    PROC MoveGridDatum()
        !Sweep across bed maintaining Z height through offsets
        FOR j FROM 9 TO 4 DO
            FOR k FROM 11 TO 1 DO
                !Move x
                PlotBedGrid(k*XGridSpacing+100),(j*YGridSpacing+100),Bed1Zread{10-j,(k+1)};
            ENDFOR
        ENDFOR
    ENDPROC


    PROC VacuumBed()

        VAR num VacOverlap:=-400;
        IF ToolNum<>5 THEN
            Home;
            Vac_Pickup;
        ELSE
            CurrentJoints:=CJointT();
            CurrentPos:=CalcRobT(CurrentJoints,tVac\WObj:=Bed1Wyong);
            IF CurrentPos.trans.x<0 AND (CurrentPos.trans.z<150) THEN
                MoveL Offs(CurrentPos,0,0,(150-CurrentPos.trans.z)),v500,z5,tVac\WObj:=Bed1Wyong;
            ELSEIF (CurrentPos.trans.z<700) THEN
                MoveL Offs(CurrentPos,0,0,(700-CurrentPos.trans.z)),v500,z5,tVac\WObj:=Bed1Wyong;
            ENDIF
        ENDIF

        pTemp:=pVacStart;
        pTemp2:=pVacStart;
        pTemp2.trans.x:=pVacStart2.trans.x;
        pTemp2.extax.eax_a:=pVacStart2.extax.eax_a;

        Vac_on;
        FOR i FROM 0 TO (Round((pVacStart.trans.y-pVacStart2.trans.y)/(-1*VacOverlap))) DO
            IF pTemp.trans.y+i*VacOverlap>pVacStart2.trans.y THEN
                MoveJ Offs(pTemp,0,i*VacOverlap,150),v500,z5,tVac\WObj:=Bed1Wyong;
                MoveL Offs(pTemp,0,i*VacOverlap,0),v50,z5,tVac\WObj:=Bed1Wyong;
                MoveL Offs(pTemp2,0,i*VacOverlap,0),v100,z5,tVac\WObj:=Bed1Wyong;
                MoveL Offs(pTemp2,0,i*VacOverlap,150),v50,fine,tVac\WObj:=Bed1Wyong;
            ENDIF
        ENDFOR

        Vac_off;

        CurrentJoints:=CJointT();
        CurrentPos:=CalcRobT(CurrentJoints,tVac\WObj:=wobj0);
        MoveL Offs(CurrentPos,0,0,800-CurrentPos.trans.z),v100,z5,tVac\WObj:=wobj0;

    ENDPROC

    PROC JointPositions()

        VAR num PolishOverlap:=450;
        pPolTemp:=pPolStart1;
        pPolTemp2:=pPolStart1;
        pPolTemp2.extax.eax_a:=pPolStart1.extax.eax_a-7500;
        pPolTemp2.trans.x:=-7500;

        pPolTemp.rot:=pPolStart1.rot;
        pPolTemp2.rot:=pPolStart1.rot;

        pPolTemp2.rot:=pPolStart2.rot;
        pPolTemp2.extax.eax_a:=pPolStart1.extax.eax_a-8500;
        CurrentJoints5:=CJointT();
        CurrentJoints6:=CalcJointT(Offs(pPolTemp2,50,(1+1)*PolishOverlap,40),tPolish\WObj:=Bed1Wyong);

    ENDPROC


    PROC RobbiePlot()

        ! !Write R
        !PlotLine 6900,1000, 6900,2000;
        !PlotArc 6900,2000,6650,1750,6900,1500;
        !PlotLine 6900,1500,6650,1000;

        !!Write O
        !PlotArc 6300,2000, 6050,1500,6300,1000;
        !PlotArc 6300,1000, 6550,1500,6300,2000;

        !!Write B
        !PlotLine 5700,1000, 5700,2000;
        !PlotArc 5700,2000,5450,1750,5700,1500;
        !PlotArc 5700,1500,5450,1250,5700,1000;

        !!Write B
        !PlotLine 5100,1000, 5100,2000;
        !PlotArc 5100,2000,4850,1750,5100,1500;
        !PlotArc 5100,1500,4850,1250,5100,1000;

        !!Write I
        !PlotLine 4500,1000, 4500,2000;

        !!Write E
        !PlotLine 3900,1000, 3900,2000;
        !PlotLine 3900,2000, 3400,2000;
        !PlotLine 3900,1500, 3400,1500;
        !PlotLine 3900,1000, 3400,1000;

        !formbox
        PlotRect 2000,500,2000,3500,6000,3500,6000,500;
        !Ferrule
        WaitTime\inpos,0.1;
        PlotCirc 2250,750,(PlotCircleD/2);
        PlotLine(2250-PlotCircleD/2-CrossHairExt),750,(2250+PlotCircleD/2+CrossHairExt),750;
        PlotLine 2250,(750-PlotCircleD/2-CrossHairExt),2250,(750+PlotCircleD/2+CrossHairExt);
        !Ferrule
        WaitTime\inpos,0.1;
        PlotCirc 2250,3250,(PlotCircleD/2);
        PlotLine(2250-PlotCircleD/2-CrossHairExt),3250,(2250+PlotCircleD/2+CrossHairExt),3250;
        PlotLine 2250,(3250-PlotCircleD/2-CrossHairExt),2250,(3250+PlotCircleD/2+CrossHairExt);
        !Grout tube Casee 4
        WaitTime\inpos,0.1;
        iCoord1x:=6000;
        iCoord1y:=2000;
        iAngle:=0;
        PlotRect iCoord1x-GroutWidth/2*Sin(iAngle)-GroutHeight*Cos(iAngle),iCoord1y+GroutHeight*Sin(iAngle)-GroutWidth/2*Cos(iAngle),iCoord1x+GroutWidth/2*Sin(iAngle)-GroutHeight*Cos(iAngle),iCoord1y+GroutHeight*Sin(iAngle)+GroutWidth/2*Cos(iAngle),iCoord1x+GroutWidth/2*Sin(iAngle),iCoord1y+GroutWidth/2*Cos(iAngle),iCoord1x-GroutWidth/2*Sin(iAngle),iCoord1y-GroutWidth/2*Cos(iAngle);

        !Lifting points 180 angle
        WaitTime\inpos,0.1;
        TriangleAngle:=180;
        iCoord1x:=5000;
        iCoord1y:=3500;
        PlotLine iCoord1x-TriangleHeight*Sin(TriangleAngle),iCoord1y-TriangleHeight*Cos(TriangleAngle),iCoord1x-TriangleBase/2*Cos(TriangleAngle),iCoord1y+TriangleBase/2*Sin(TriangleAngle);
        PlotLine iCoord1x-TriangleBase/2*Cos(TriangleAngle),iCoord1y+TriangleBase/2*Sin(TriangleAngle),iCoord1x+TriangleBase/2*Cos(TriangleAngle),iCoord1y-TriangleBase/2*Sin(TriangleAngle);
        PlotLine iCoord1x+TriangleBase/2*Cos(TriangleAngle),iCoord1y-TriangleBase/2*Sin(TriangleAngle),iCoord1x-TriangleHeight*Sin(TriangleAngle),iCoord1y-TriangleHeight*Cos(TriangleAngle);
        !Lifting points 180 angle
        WaitTime\inpos,0.1;
        TriangleAngle:=180;
        iCoord1x:=3000;
        iCoord1y:=3500;
        PlotLine iCoord1x-TriangleHeight*Sin(TriangleAngle),iCoord1y-TriangleHeight*Cos(TriangleAngle),iCoord1x-TriangleBase/2*Cos(TriangleAngle),iCoord1y+TriangleBase/2*Sin(TriangleAngle);
        PlotLine iCoord1x-TriangleBase/2*Cos(TriangleAngle),iCoord1y+TriangleBase/2*Sin(TriangleAngle),iCoord1x+TriangleBase/2*Cos(TriangleAngle),iCoord1y-TriangleBase/2*Sin(TriangleAngle);
        PlotLine iCoord1x+TriangleBase/2*Cos(TriangleAngle),iCoord1y-TriangleBase/2*Sin(TriangleAngle),iCoord1x-TriangleHeight*Sin(TriangleAngle),iCoord1y-TriangleHeight*Cos(TriangleAngle);

        Plotter_Dropoff;

    ENDPROC

    PROC PolishDemo()
        IF ToolNum<>6 THEN
            Home;
            Polish_Pickup;
        ELSE
            CurrentJoints:=CJointT();
            CurrentPos:=CalcRobT(CurrentJoints,tPolish\WObj:=wobj0);
            IF CurrentPos.trans.z<600 THEN
                MoveL Offs(CurrentPos,0,0,(600-CurrentPos.trans.z)),v500,z5,tPolish;
            ENDIF
        ENDIF
        MoveJ pPolHome,v500,z5,tPolish;
        pPolTemp:=pPolStart1;
        pPolTemp2:=pPolStart1;
        pPolTemp2.extax.eax_a:=pPolStart1.extax.eax_a-7500;
        pPolTemp2.trans.x:=-7500;
        pPolTemp.rot:=pPolStart1.rot;
        pPolTemp2.rot:=pPolStart1.rot;
        FCCalib PolishLoad;
        pPolTemp.extax.eax_a:=pPolStart1.extax.eax_a;
        MoveJ Offs(pPolTemp,0,0,100),v500,z5,tPolish\WObj:=Bed1Wyong;
        Pol_on;
        MoveL Offs(pPolTemp,0,0,50),v100,fine,tPolish\WObj:=Bed1Wyong;
        myForceVector:=FCGetForce(\Tool:=tPolish);
        FCPress1LStart Offs(pPolTemp,-25,0,55),v10,\Fz:=120,15,\ForceChange:=50\PosSupvDist:=125,z5,tPolish\WObj:=Bed1Wyong;
        pPolTemp2.extax.eax_a:=pPolStart2.extax.eax_a-300;
        FCPressL Offs(pPolTemp2,-300,0,-15),v100,130,fine,tPolish\WObj:=Bed1Wyong;
        FCPressEnd Offs(pPolTemp2,-300,0,75),v50,\DeactOnly,tPolish\WObj:=Bed1Wyong;
        CurrentJoints:=CJointT();
        CurrentPos:=CalcRobT(CurrentJoints,tPolish\WObj:=Bed1Wyong);
        MoveJ Offs(Reltool(CurrentPos,0,0,-100),0,450,0),v100,fine,tPolish\WObj:=Bed1Wyong;
        Pol_off;
        Polish_Dropoff;
    ENDPROC



    PROC BedGrid()

        !        MoveJ Offs(p10Maps,500*(1-1)+2000*(1-1),650*(1-1),50),v500,z5,tTCMaster\WObj:=Bed1Wyong;
        !        MoveL Offs(p10Maps,500*(1-1)+2000*(1-1),650*(1-1),0),v500,fine,tTCMaster\WObj:=Bed1Wyong;
        !        Stop;
        !        MoveL Offs(p10Maps,500*(1-1)+2000*(1-1),650*(1-1),50),v500,z5,tTCMaster\WObj:=Bed1Wyong;
        !        Stop;

        FOR i FROM 1 TO 5 DO
            !Move EAX
            FOR k FROM 1 TO 4 DO
                !Move x
                FOR j FROM 1 TO 4 DO
                    !Move y
                    IF 500*(k-1)+2000*(i-1)<8001 THEN
                        p10maps.extax.eax_a:=Bed1Wyong.uframe.trans.x+p10Maps.trans.x-500*(k-1)-2000*(i-1);
                        IF p10maps.extax.eax_a>10150 THEN
                            p10maps.extax.eax_a:=10100;
                        ENDIF
                        IF p10maps.extax.eax_a<1000 THEN
                            p10maps.extax.eax_a:=1000;
                        ENDIF

                        !MoveJ Offs(p10Maps,-500*(k-1)-2000*(i-1),650*(j-1),50),v500,z5,tTCMaster\WObj:=Bed1Wyong;
                        !MoveL Offs(p10Maps,-500*(k-1)-2000*(i-1),650*(j-1),0),v500,fine,tTCMaster\WObj:=Bed1Wyong;
                        !TPReadNum BedZread,"Enter Z reading";
                        !BedZreads{5-j,((i-1)*4+k)}:=BedZread;
                        BedZpos{5-j,((i-1)*4+k),1}:=p10Maps.trans.x-500*(k-1)-2000*(i-1);
                        BedZpos{5-j,((i-1)*4+k),2}:=p10maps.trans.y+650*(j-1);
                        !MoveL Offs(p10Maps,-500*(k-1)-2000*(i-1),650*(j-1),50),v500,z5,tTCMaster\WObj:=Bed1Wyong;
                    ENDIF

                ENDFOR
            ENDFOR
        ENDFOR
        Stop;

    ENDPROC


    PROC ClearBedZ()

        FOR i FROM 1 TO 4 DO
            !Move EAX
            FOR k FROM 1 TO 24 DO
                !Move x
                BedZreads{i,k}:=0;
                BedZpos{i,k,1}:=0;
                BedZpos{i,k,2}:=0;
            ENDFOR
        ENDFOR

    ENDPROC




    PROC BHTestTask()
        TPErase;
        TPWrite "BH Test Task";
        TPWrite "Press Play to confirm and start task";
        Stop;

        TPErase;
        TPWrite "Starting BH Test Task...";

        Heli_Pickup;
        MoveJ Offs(ptHeli,0,0,1000),v500,fine,tHeli;
        TPWrite "Helicopter tool at 1000mm above pickup";
        WaitTime 2;

        Heli_Dropoff;
        TPWrite "Helicopter tool dropped off";

        Polish_Pickup;
        MoveJ Offs(ptPolish,0,0,1000),v500,fine,tPolish;
        TPWrite "Polisher tool at 1000mm above pickup";
        WaitTime 2;

        Polish_Dropoff;
        TPWrite "Polisher tool dropped off";

        Home;
        TPWrite "BH Test Task Complete";

    ERROR
        RAISE ;
    ENDPROC



    PROC Datum()
        ! Datum - draws small circle at Bed1Wyong origin (0,0)
        ! Generated by Onyx Toolpath Generator
        VAR robtarget pDatumCenter;
        VAR robtarget pDatumCircle;
        VAR num DatumZ:=300;
        VAR num DatumRadius:=100;
        VAR num SafeZ:=500;
        VAR num i;

        TPWrite "Datum: ToolNum=" \Num:=ToolNum;
        IF ToolNum<>4 THEN
            TPWrite "No plotter! Will pickup plotter.";
            Stop;
            Home;
            Plotter_Pickup;
        ELSE
            CurrentJoints:=CJointT();
            CurrentPos:=CalcRobT(CurrentJoints,tPlotter\WObj:=wobj0);
            IF CurrentPos.trans.z<600 THEN
                MoveL Offs(CurrentPos,0,0,(600-CurrentPos.trans.z)),v500,z5,tPlotter;
            ENDIF
        ENDIF

        ConfL\Off;
        ConfJ\Off;

        pDatumCenter:=[[0,0,DatumZ],[0,0,1,0],[0,0,0,0],[0,9E+09,9E+09,9E+09,9E+09,9E+09]];
        pDatumCenter.rot:=OrientZYX(-90,0,180);
        pDatumCenter.extax.eax_a:=6500;

        TPWrite "Datum: Drawing circle at origin";
        TPWrite "Press Play to continue";
        Stop;

        pDatumCircle:=pDatumCenter;
        pDatumCircle.trans.z:=SafeZ;
        MoveJ pDatumCircle,v500,z5,tPlotter\WObj:=Bed1Wyong;

        pDatumCircle.trans.x:=DatumRadius;
        pDatumCircle.trans.z:=DatumZ;
        MoveJ pDatumCircle,v500,z5,tPlotter\WObj:=Bed1Wyong;

        FOR i FROM 1 TO 8 DO
            pDatumCircle.trans.x:=DatumRadius*Cos(i*45);
            pDatumCircle.trans.y:=DatumRadius*Sin(i*45);
            MoveJ pDatumCircle,v100,fine,tPlotter\WObj:=Bed1Wyong;
        ENDFOR

        pDatumCircle.trans.x:=0;
        pDatumCircle.trans.y:=0;
        pDatumCircle.trans.z:=DatumZ;
        MoveJ pDatumCircle,v100,fine,tPlotter\WObj:=Bed1Wyong;

        TPWrite "Plotter at datum center (0,0)";
        TPWrite "Press Play to return tool";
        Stop;

        pDatumCircle.trans.z:=SafeZ;
        MoveJ pDatumCircle,v500,z5,tPlotter\WObj:=Bed1Wyong;

        ConfL\On;
        ConfJ\On;

        Plotter_Dropoff;
        Home;

        TPWrite "Datum Complete";
    ERROR
        RAISE;
    ENDPROC


    PROC PyHeli()
        ! PyHeli - Helicopter serpentine pattern
        ! Workzone: panel
        ! Force Control DISABLED (dummy run)
        ! Generated by Onyx Toolpath Generator

        VAR robtarget pHeliPos;
        VAR robtarget pHeliEnd;
        VAR num HeliZ:=450;
        VAR num SafeZ:=500;

        ! Workspace bounds (with offsets applied)
        VAR num WorkMinX:=2200;
        VAR num WorkMaxX:=7850;
        VAR num WorkMinY:=200;
        VAR num WorkMaxY:=2200;

        ! Pattern parameters
        VAR num StepSize:=450;
        VAR num SweepDir:=1;
        VAR num StepDir:=-1;
        VAR num CurrentY:=2200;
        VAR num CurrentX:=2200;
        VAR num NextY;
        VAR num NextX;
        VAR num StartX;
        VAR num EndX;
        VAR num StartY;
        VAR num EndY;

        ! Speed and blade parameters
        VAR num HeliSpeed:=100;
        VAR num HeliAngle:=1;
        VAR speeddata vHeliTravel:=[500,15,2000,15];
        VAR num NumPasses;
        ! Force control disabled

        NumPasses:=Trunc(Abs(WorkMaxY-WorkMinY)/StepSize)+1;

        TPWrite "PyHeli: Serpentine Pattern";
        TPWrite "Work Area (7850,2200) to (2200,200)";
        TPWrite "Passes=" \Num:=NumPasses;
        TPWrite "Step=" \Num:=StepSize;
        TPWrite "Force=OFF (dummy)";

        IF ToolNum<>2 THEN
            TPWrite "PyHeli: ToolNum<>2, need pickup";
            Stop;
            Home;
            Heli_Pickup;
        ELSE
            CurrentJoints:=CJointT();
            CurrentPos:=CalcRobT(CurrentJoints,tHeli\WObj:=Bed1Wyong);
            IF CurrentPos.trans.z<SafeZ THEN
                MoveL Offs(CurrentPos,0,0,(SafeZ-CurrentPos.trans.z)),v500,z5,tHeli\WObj:=Bed1Wyong;
            ENDIF
        ENDIF

        ! Set start/end based on sweep direction
        IF SweepDir=1 THEN
            StartX:=WorkMinX;
            EndX:=WorkMaxX;
        ELSE
            StartX:=WorkMaxX;
            EndX:=WorkMinX;
        ENDIF

        ! Set initial position with fixed orientation
        pHeliPos:=[[0,0,HeliZ],OrientZYX(0,0,180),[0,0,0,0],[0,9E+09,9E+09,9E+09,9E+09,9E+09]];

        ! Move to row start above surface (HOVER)
        pHeliPos.trans.x:=-StartX;
        pHeliPos.trans.y:=CurrentY;
        pHeliPos.trans.z:=SafeZ;
        pHeliPos.extax.eax_a:=Bed1Wyong.uframe.trans.x-StartX;
        MoveJ pHeliPos,v500,z5,tHeli\WObj:=Bed1Wyong;

        ! Disable configuration tracking for serpentine movements
        ConfL\Off;
        ConfJ\Off;

        ! Home stepper before setting blade angle (ensures StepperPos is valid)
        TPWrite "Homing blade stepper...";
        Heli_Stepper_Home;
        TPWrite "Stepper homed";

        ! Set blade angle while hovering
        TPWrite "Setting blade angle to " \Num:=HeliAngle;
        HeliBlade_Angle HeliAngle;
        WaitTime 2;
        TPWrite "Blade angle set";

        ! No force calibration needed

        TPWrite "Hovering over workspace - Press Play to start";
        Stop;

        ! Start blade rotation BEFORE lowering
        TPWrite "Starting blade rotation...";
        HeliBladeSpeed HeliSpeed,"FWD";
        WaitTime 1;

        ! Lower to working height
        TPWrite "Lowering to work surface...";
        pHeliPos.trans.z:=HeliZ;
        MoveL pHeliPos,v50,fine,tHeli\WObj:=Bed1Wyong;

        ! No force control - dummy run

        ! Set up end position for first sweep
        pHeliEnd:=pHeliPos;
        pHeliEnd.trans.x:=-EndX;
        pHeliEnd.extax.eax_a:=Bed1Wyong.uframe.trans.x-EndX;

        ! ========== PASS 1: X-direction sweeps (stepping in Y) ===========
        WHILE TRUE DO
            ! === SWEEP X (full length) ===
            MoveL pHeliEnd,vHeliTravel,fine,tHeli\WObj:=Bed1Wyong;

            ! No force ramping in dummy mode

            ! Calculate next row
            NextY:=CurrentY+(StepDir*StepSize);

            ! Check if pass complete
            IF (StepDir=1 AND NextY>WorkMaxY) OR (StepDir=-1 AND NextY<WorkMinY) THEN
                EXIT;
            ENDIF

            ! Clamp to bounds
            IF NextY>WorkMaxY THEN
                NextY:=WorkMaxY;
            ELSEIF NextY<WorkMinY THEN
                NextY:=WorkMinY;
            ENDIF

            ! Step to next Y row
            pHeliEnd.trans.y:=NextY;
            MoveL pHeliEnd,vHeliTravel,fine,tHeli\WObj:=Bed1Wyong;
            CurrentY:=NextY;

            ! Flip sweep direction
            SweepDir:=-SweepDir;
            IF SweepDir=1 THEN
                StartX:=WorkMinX;
                EndX:=WorkMaxX;
            ELSE
                StartX:=WorkMaxX;
                EndX:=WorkMinX;
            ENDIF

            ! Set up end position for next sweep
            pHeliEnd.trans.x:=-EndX;
            pHeliEnd.extax.eax_a:=Bed1Wyong.uframe.trans.x-EndX;
        ENDWHILE

        ! ========== PASS 2: Y-direction sweeps (stepping in X) ==========
        TPWrite "=== PASS 2 START ===";

        ! Reset for Y-direction passes - start from current position
        CurrentX:=Abs(pHeliEnd.trans.x);
        TPWrite "Pass2: CurrentX=" \Num:=CurrentX;
        TPWrite "Pass2: CurrentY=" \Num:=CurrentY;
        TPWrite "Pass2: WorkMinX=" \Num:=WorkMinX;
        TPWrite "Pass2: WorkMaxX=" \Num:=WorkMaxX;

        ! Determine step direction based on where Pass 1 ended
        ! At high X, step toward low X; at low X, step toward high X
        IF CurrentX>((WorkMinX+WorkMaxX)/2) THEN
            StepDir:=-1;
            TPWrite "Pass2: StepDir=-1 (toward MinX)";
        ELSE
            StepDir:=1;
            TPWrite "Pass2: StepDir=+1 (toward MaxX)";
        ENDIF

        ! Determine sweep direction based on where Pass 1 ended (which Y edge)
        IF CurrentY>((WorkMinY+WorkMaxY)/2) THEN
            SweepDir:=1;
            StartY:=WorkMaxY;
            EndY:=WorkMinY;
            TPWrite "Pass2: Sweep MinY first";
        ELSE
            SweepDir:=-1;
            StartY:=WorkMinY;
            EndY:=WorkMaxY;
            TPWrite "Pass2: Sweep MaxY first";
        ENDIF

        TPWrite "Pass2: EndY=" \Num:=EndY;

        ! First Y sweep from current position
        TPWrite "Pass2: First Y sweep...";
        pHeliEnd.trans.y:=EndY;
        MoveL pHeliEnd,vHeliTravel,fine,tHeli\WObj:=Bed1Wyong;
        TPWrite "Pass2: First Y sweep done";

        TPWrite "Pass2: Entering X-step loop";

        WHILE TRUE DO
            ! Calculate next column
            NextX:=CurrentX+(StepDir*StepSize);
            TPWrite "Pass2: NextX=" \Num:=NextX;

            ! Check if pass complete (no more columns to step to)
            IF (StepDir=1 AND NextX>WorkMaxX) OR (StepDir=-1 AND NextX<WorkMinX) THEN
                TPWrite "Pass2: EXIT - NextX out of bounds";
                ! No force control end needed
                EXIT;
            ENDIF

            ! Clamp to bounds
            IF NextX>WorkMaxX THEN
                NextX:=WorkMaxX;
            ELSEIF NextX<WorkMinX THEN
                NextX:=WorkMinX;
            ENDIF

            ! Step to next X column
            TPWrite "Pass2: Step to X=" \Num:=NextX;
            pHeliEnd.trans.x:=-NextX;
            pHeliEnd.extax.eax_a:=Bed1Wyong.uframe.trans.x-NextX;
            MoveL pHeliEnd,vHeliTravel,fine,tHeli\WObj:=Bed1Wyong;
            CurrentX:=NextX;

            ! Flip sweep direction for next Y sweep
            SweepDir:=-SweepDir;
            IF SweepDir=1 THEN
                EndY:=WorkMinY;
            ELSE
                EndY:=WorkMaxY;
            ENDIF

            ! Set up end position and sweep Y
            TPWrite "Pass2: Sweep Y to " \Num:=EndY;
            pHeliEnd.trans.y:=EndY;
            MoveL pHeliEnd,vHeliTravel,fine,tHeli\WObj:=Bed1Wyong;
        ENDWHILE
        TPWrite "=== PASS 2 COMPLETE ===";

        ! === LIFT OFF BED ===
        pHeliPos.trans.z:=SafeZ;
        MoveL pHeliPos,v100,z5,tHeli\WObj:=Bed1Wyong;

        ! === STOP BLADE ROTATION ===
        HeliBladeSpeed 0,"FWD";
        WaitTime\InPos,3;

        ConfL\On;
        ConfJ\On;

        ! === PACKAWAY ===
        Heli_Dropoff;
        Home;

        TPWrite "PyHeli Complete";
    ERROR
        HeliBladeSpeed 0,"FWD";
        RAISE;
    ENDPROC


    PROC PyVac()
        ! PyVac - Vacuum procedure with serpentine pattern
        ! Workzone: bed
        ! Generated by Onyx Toolpath Generator

        VAR robtarget pVacPos;
        VAR robtarget pVacEnd;
        VAR num VacZ:=280;
        VAR num SafeZ:=300;

        ! Force control parameters
        VAR num VacForce:=50;
        VAR num VacZMin:=-20;
        VAR num VacZMax:=50;
        VAR num VacZRange:=70;

        ! Workspace bounds (with offsets applied)
        VAR num WorkMinX:=0;
        VAR num WorkMaxX:=8500;
        VAR num WorkMinY:=0;
        VAR num WorkMaxY:=1650;

        ! Pattern parameters
        VAR num StepSize:=300;
        VAR num SweepDir:=-1;
        VAR num YStepDir:=-1;
        VAR num CurrentY:=1650;
        VAR num NextY;
        VAR num StartX;
        VAR num EndX;

        VAR speeddata vVac:=[200,30,2000,15];
        VAR num NumPasses;

        NumPasses:=Trunc(Abs(WorkMaxY-WorkMinY)/StepSize)+1;

        TPWrite "PyVac: Serpentine Pattern";
        TPWrite "Work Area (8500,1650) to (0,0)";
        TPWrite "Passes=" \Num:=NumPasses;
        TPWrite "Step=" \Num:=StepSize;
        TPWrite "Speed=" \Num:=200;

        IF ToolNum<>5 THEN
            TPWrite "PyVac: ToolNum<>5, need pickup";
            TPWrite "PyVac: ToolNum=" \Num:=ToolNum;
            TPWrite "PyVac: Calling Vac_Pickup...";
            Stop;
            Vac_Pickup;
            TPWrite "PyVac: Vac_Pickup complete";
        ELSE
            CurrentJoints:=CJointT();
            CurrentPos:=CalcRobT(CurrentJoints,tVac\WObj:=Bed1Wyong);
            IF CurrentPos.trans.z<SafeZ THEN
                MoveL Offs(CurrentPos,0,0,(SafeZ-CurrentPos.trans.z)),v500,z5,tVac\WObj:=Bed1Wyong;
            ENDIF
        ENDIF

        ConfL\Off;
        ConfJ\Off;

        pVacPos:=[[0,0,VacZ],[0.00615322,-0.709926,0.704246,-0.00239206],[1,-1,0,0],[0,9E+09,9E+09,9E+09,9E+09,9E+09]];

        TPWrite "Press Play to start";
        Stop;

        Vac_on;

        ! Main vacuum loop - always sweep right to left, lift and return
        WHILE TRUE DO
            ! Move to row start above work surface (right side)
            pVacPos.trans.x:=-WorkMaxX;
            pVacPos.trans.y:=CurrentY;
            pVacPos.trans.z:=VacZMax;
            pVacPos.extax.eax_a:=Bed1Wyong.uframe.trans.x-WorkMaxX;
            MoveL pVacPos,vVac,fine,tVac\WObj:=Bed1Wyong;

            ! Set up end position
            pVacEnd:=pVacPos;
            pVacEnd.trans.x:=-WorkMinX;
            pVacEnd.trans.z:=VacZ;
            pVacEnd.extax.eax_a:=Bed1Wyong.uframe.trans.x-WorkMinX;

            ! Sweep right to left
            pVacPos.trans.z:=VacZ;
            MoveL pVacPos,vVac,fine,tVac\WObj:=Bed1Wyong;
            MoveL pVacEnd,vVac,z5,tVac\WObj:=Bed1Wyong;

            ! Calculate next row
            NextY:=CurrentY+(YStepDir*StepSize);

            ! Check if pattern complete
            IF (YStepDir=1 AND NextY>WorkMaxY) OR (YStepDir=-1 AND NextY<WorkMinY) THEN
                ! Pattern complete
                EXIT;
            ENDIF

            ! Clamp to bounds for partial last step
            IF NextY>WorkMaxY THEN
                NextY:=WorkMaxY;
            ELSEIF NextY<WorkMinY THEN
                NextY:=WorkMinY;
            ENDIF

            ! Lift off work surface (already lifted by FCPressEnd)
            pVacPos.trans.z:=SafeZ;
            pVacPos.trans.x:=-WorkMinX;
            pVacPos.extax.eax_a:=Bed1Wyong.uframe.trans.x-WorkMinX;
            MoveL pVacPos,v500,z5,tVac\WObj:=Bed1Wyong;

            ! Return to start X (right side) at safe height, step to next Y
            pVacPos.trans.x:=-WorkMaxX;
            pVacPos.trans.y:=NextY;
            pVacPos.extax.eax_a:=Bed1Wyong.uframe.trans.x-WorkMaxX;
            MoveL pVacPos,v500,z5,tVac\WObj:=Bed1Wyong;

            CurrentY:=NextY;
        ENDWHILE

        Vac_off;

        pVacPos.trans.z:=SafeZ;
        MoveL pVacPos,v100,z5,tVac\WObj:=Bed1Wyong;

        ConfL\On;
        ConfJ\On;

        Vac_Dropoff;
        Home;

        TPWrite "PyVac Complete";
    ERROR
        Vac_off;
        RAISE;
    ENDPROC


    PROC PyPolish()
        ! PyPolish - Polisher serpentine with force control
        ! Workzone: bed
        ! Generated by Onyx Toolpath Generator

        VAR robtarget pPolPos;
        VAR robtarget pPolEnd;
        VAR num PolZ:=300;
        VAR num SafeZ:=300;

        ! Force control parameters
        VAR num StartForce:=300;
        VAR num MotionForce:=300;
        VAR num ForceChange:=100;
        VAR num PosSupvDist:=100;

        ! Workspace bounds (with offsets applied)
        VAR num WorkMinX:=0;
        VAR num WorkMaxX:=8500;
        VAR num WorkMinY:=0;
        VAR num WorkMaxY:=1650;

        ! Pattern parameters
        VAR num StepSize:=300;
        VAR num SweepDir:=1;
        VAR num YStepDir:=-1;
        VAR num CurrentY:=1650;
        VAR num NextY;
        VAR num StartX;
        VAR num EndX;

        VAR speeddata vPolApproach:=[20,30,2000,15];
        VAR speeddata vPolRetract:=[50,30,2000,15];
        VAR speeddata vPolTravel:=[100,30,2000,15];
        VAR num NumPasses;

        NumPasses:=Trunc(Abs(WorkMaxY-WorkMinY)/StepSize)+1;

        TPWrite "PyPolish: Serpentine Pattern";
        TPWrite "Work Area (8500,1650) to (0,0)";
        TPWrite "Passes=" \Num:=NumPasses;
        TPWrite "Step=" \Num:=StepSize;
        TPWrite "Force=" \Num:=MotionForce;

        IF ToolNum<>6 THEN
            TPWrite "PyPolish: ToolNum<>6, need pickup";
            Stop;
            Home;
            Polish_Pickup;
        ELSE
            CurrentJoints:=CJointT();
            CurrentPos:=CalcRobT(CurrentJoints,tPolish\WObj:=Bed1Wyong);
            IF CurrentPos.trans.z<SafeZ THEN
                MoveL Offs(CurrentPos,0,0,(SafeZ-CurrentPos.trans.z)),v500,z5,tPolish\WObj:=Bed1Wyong;
            ENDIF
        ENDIF

        ConfL\Off;
        ConfJ\Off;

        ! Set start/end based on sweep direction
        IF SweepDir=1 THEN
            StartX:=WorkMinX;
            EndX:=WorkMaxX;
        ELSE
            StartX:=WorkMaxX;
            EndX:=WorkMinX;
        ENDIF

        ! Set initial position with fixed orientation (facing +X direction)
        pPolPos:=[[0,0,PolZ],OrientZYX(0,0,180),[1,-1,-1,0],[0,9E+09,9E+09,9E+09,9E+09,9E+09]];

        ! Calibrate force control
        FCCalib PolishLoad;

        TPWrite "Press Play to start";
        Stop;

        ! Move to row start above surface
        pPolPos.trans.x:=-StartX;
        pPolPos.trans.y:=CurrentY;
        pPolPos.trans.z:=SafeZ;
        pPolPos.extax.eax_a:=Bed1Wyong.uframe.trans.x-StartX;
        MoveL pPolPos,vPolTravel,z5,tPolish\WObj:=Bed1Wyong;

        ! Lower to approach height
        pPolPos.trans.z:=PolZ+50;
        MoveL pPolPos,vPolApproach,fine,tPolish\WObj:=Bed1Wyong;

        ! Turn on polisher and wait for spin-up
        Pol_off;
        WaitTime 0.2;
        Pol_on;
        WaitTime 1.0;

        ! Set up end position for first sweep
        pPolEnd:=pPolPos;
        pPolEnd.trans.x:=-EndX;
        pPolEnd.trans.z:=PolZ;
        pPolEnd.extax.eax_a:=Bed1Wyong.uframe.trans.x-EndX;

        ! Start force control
        FCPress1LStart Offs(pPolPos,0,0,25),vPolApproach,\Fz:=StartForce,15,\ForceChange:=ForceChange\PosSupvDist:=PosSupvDist,z5,tPolish\WObj:=Bed1Wyong;

        ! Main polisher loop - stays in contact during serpentine
        WHILE TRUE DO
            ! === SWEEP X (full length) ===
            FCPressL pPolEnd,vPolTravel,MotionForce,fine,tPolish\WObj:=Bed1Wyong;

            ! Calculate next row
            NextY:=CurrentY+(YStepDir*StepSize);

            ! Check if pattern complete
            IF (YStepDir=1 AND NextY>WorkMaxY) OR (YStepDir=-1 AND NextY<WorkMinY) THEN
                FCPressEnd Offs(pPolEnd,0,0,50),vPolRetract,\DeactOnly,tPolish\WObj:=Bed1Wyong;
                Pol_off;
                EXIT;
            ENDIF

            ! Clamp to bounds
            IF NextY>WorkMaxY THEN
                NextY:=WorkMaxY;
            ELSEIF NextY<WorkMinY THEN
                NextY:=WorkMinY;
            ENDIF

            ! Step to next Y row (still in force control)
            pPolEnd.trans.y:=NextY;
            FCPressL pPolEnd,vPolTravel,MotionForce,fine,tPolish\WObj:=Bed1Wyong;
            CurrentY:=NextY;

            ! Flip sweep direction
            SweepDir:=-SweepDir;
            IF SweepDir=1 THEN
                StartX:=WorkMinX;
                EndX:=WorkMaxX;
            ELSE
                StartX:=WorkMaxX;
                EndX:=WorkMinX;
            ENDIF

            ! Set up end position for next sweep
            pPolEnd.trans.x:=-EndX;
            pPolEnd.extax.eax_a:=Bed1Wyong.uframe.trans.x-EndX;
        ENDWHILE

        ! Return to safe height
        pPolPos.trans.z:=SafeZ;
        MoveL pPolPos,vPolTravel,z5,tPolish\WObj:=Bed1Wyong;

        ConfL\On;
        ConfJ\On;

        Polish_Dropoff;
        Home;

        TPWrite "PyPolish Complete";
    ERROR
        Pol_off;
        RAISE;
    ENDPROC


    PROC PyVibScreed()
        ! PyVibScreed - Vibrating Screed with Panel workzone parameters
        ! Workzone: Panel
        ! Panel: X=2200 to 7850, Y=200, Z=150
        ! Panel Start/Finish Offset: 200 mm
        ! Actual travel: X=2000 to 8050
        ! Global Z Offset: 300 mm
        ! Screed Z Offset: 4 mm
        ! Working Z: 454 mm
        ! Speed: 50 mm/s
        ! Angle: 11°
        ! Generated by Onyx Toolpath Generator

        VAR robtarget pScreedPos;
        VAR robtarget pScreedEnd;
        VAR num ScrStartX:=2000;
        VAR num ScrEndX:=8050;
        VAR num ScrY:=200;
        VAR num WorkZ:=454;
        VAR num SafeZ:=500;
        VAR num ScrAoffset:=11;
        VAR speeddata vScreed:=[50,30,2000,15];

        TPWrite "PyVibScreed: Panel Workzone";
        TPWrite "Start X=" \Num:=ScrStartX;
        TPWrite "End X=" \Num:=ScrEndX;
        TPWrite "Y=" \Num:=ScrY;
        TPWrite "Work Z=" \Num:=WorkZ;
        TPWrite "Speed=" \Num:=50;
        TPWrite "Angle=" \Num:=ScrAoffset;

        CurrentJoints:=CJointT();
        CurrentPos:=CalcRobT(CurrentJoints,tVS\WObj:=Bed1Wyong);

        IF ToolNum<>3 THEN
            TPWrite "PyVibScreed: ToolNum<>3, need pickup";
            Stop;
            Home;
            VS_Pickup;
        ELSEIF (CurrentPos.trans.z<SafeZ) THEN
            MoveL Offs(CurrentPos,0,0,(SafeZ-CurrentPos.trans.z)),v200,z5,tVS\WObj:=Bed1Wyong;
        ENDIF

        ! Set up start position - use pVSstart as template for rotation
        pScreedPos:=pVSstart;
        pScreedPos.trans.x:=-ScrStartX;
        pScreedPos.trans.y:=ScrY;
        pScreedPos.trans.z:=SafeZ;
        pScreedPos.extax.eax_a:=Bed1Wyong.uframe.trans.x-ScrStartX+700;

        ! Set up end position
        pScreedEnd:=pScreedPos;
        pScreedEnd.trans.x:=-ScrEndX;
        pScreedEnd.trans.z:=WorkZ;
        pScreedEnd.extax.eax_a:=Bed1Wyong.uframe.trans.x-ScrEndX+700;

        ! Move to start position at safe height (holding high)
        MoveL pScreedPos,v500,fine,tVS\WObj:=Bed1Wyong;

        ! Drop down to approach height (100mm above work)
        pScreedPos.trans.z:=WorkZ+100;
        MoveL RelTool(pScreedPos,0,0,0\Ry:=ScrAoffset),v200,fine,tVS\WObj:=Bed1Wyong;

        ! Start vibrator
        VS_on;

        ! Lower to working Z
        pScreedPos.trans.z:=WorkZ;
        MoveL RelTool(pScreedPos,0,0,0\Ry:=ScrAoffset),v50,z5,tVS\WObj:=Bed1Wyong;

        ! Screed across panel
        MoveL RelTool(pScreedEnd,0,0,0\Ry:=ScrAoffset),vScreed,z5,tVS\WObj:=Bed1Wyong;

        ! Lift off at end
        pScreedEnd.trans.z:=WorkZ+100;
        MoveL RelTool(pScreedEnd,0,0,0\Ry:=ScrAoffset),v100,z5,tVS\WObj:=Bed1Wyong;

        VS_off;

        ! Return to safe height
        pScreedEnd.trans.z:=SafeZ;
        MoveL pScreedEnd,v200,z5,tVS\WObj:=Bed1Wyong;

        VS_Dropoff;

        TPWrite "PyVibScreed Complete";
    ENDPROC


    PROC PyPan()
        ! Python-generated Pan procedure
        ! Serpentine pattern over Panel workzone

        VAR robtarget pPanPos;
        VAR robtarget pPanEnd;
        VAR robtarget CurrentPos;
        VAR jointtarget CurrentJoints;

        ! Workspace bounds (Panel)
        CONST num WorkMinX:=2200;
        CONST num WorkMaxX:=7850;
        CONST num WorkMinY:=200;
        CONST num WorkMaxY:=2200;
        CONST num PanZ:=451;
        CONST num SafeZ:=751;

        ! Pattern parameters
        VAR num StepSize:=500;
        VAR num SweepDir:=1;
        VAR num StepDir:=-1;
        VAR num CurrentY:=2200;
        VAR num CurrentX:=2200;
        VAR num NextY;
        VAR num NextX;
        VAR num StartX;
        VAR num EndX;
        VAR num StartY;
        VAR num EndY;

        ! Speed and blade parameters
        VAR num PanSpeed:=140;
        VAR num PanAngle:=0;  ! Pan always uses 0 blade angle
        VAR speeddata vPanTravel:=[500,30,2000,15];
        VAR num NumPasses;

        NumPasses:=Trunc(Abs(WorkMaxY-WorkMinY)/StepSize)+1;

        TPWrite "PyPan: Serpentine Pattern";
        TPWrite "Work Area (7850,2200) to (2200,200)";
        TPWrite "Passes=" \Num:=NumPasses;
        TPWrite "Step=" \Num:=StepSize;

        IF ToolNum<>2 THEN
            TPWrite "PyPan: ToolNum<>2, need pickup";
            Stop;
            Home;
            Heli_Pickup;
        ELSE
            CurrentJoints:=CJointT();
            CurrentPos:=CalcRobT(CurrentJoints,tHeli\WObj:=Bed1Wyong);
            IF CurrentPos.trans.z<SafeZ THEN
                MoveL Offs(CurrentPos,0,0,(SafeZ-CurrentPos.trans.z)),v500,z5,tHeli\WObj:=Bed1Wyong;
            ENDIF
        ENDIF

        ! Set start/end based on sweep direction
        IF SweepDir=1 THEN
            StartX:=WorkMinX;
            EndX:=WorkMaxX;
        ELSE
            StartX:=WorkMaxX;
            EndX:=WorkMinX;
        ENDIF

        ! Set initial position with fixed orientation
        pPanPos:=[[0,0,PanZ],OrientZYX(0,0,180),[0,0,0,0],[0,9E+09,9E+09,9E+09,9E+09,9E+09]];

        ! Move to row start above surface
        pPanPos.trans.x:=-StartX;
        pPanPos.trans.y:=CurrentY;
        pPanPos.trans.z:=SafeZ;
        pPanPos.extax.eax_a:=Bed1Wyong.uframe.trans.x-StartX;
        MoveJ pPanPos,v500,z5,tHeli\WObj:=Bed1Wyong;

        TPWrite "Press Play to start";
        Stop;

        ! Disable configuration tracking for serpentine movements
        ConfL\Off;
        ConfJ\Off;

        ! Lower to working height
        pPanPos.trans.z:=PanZ;
        MoveL pPanPos,v50,fine,tHeli\WObj:=Bed1Wyong;

        ! Start blade rotation
        HeliBladeSpeed PanSpeed,"FWD";
        WaitTime\InPos,3;

        ! Set up end position for first sweep
        pPanEnd:=pPanPos;
        pPanEnd.trans.x:=-EndX;
        pPanEnd.extax.eax_a:=Bed1Wyong.uframe.trans.x-EndX;

        ! ========== PASS 1: X-direction sweeps (stepping in Y) ===========
        WHILE TRUE DO
            ! === SWEEP X (full length) ===
            MoveL pPanEnd,vPanTravel,z5,tHeli\WObj:=Bed1Wyong;

            ! Calculate next row
            NextY:=CurrentY+(StepDir*StepSize);

            ! Check if pass complete
            IF (StepDir=1 AND NextY>WorkMaxY) OR (StepDir=-1 AND NextY<WorkMinY) THEN
                EXIT;
            ENDIF

            ! Clamp to bounds
            IF NextY>WorkMaxY THEN
                NextY:=WorkMaxY;
            ELSEIF NextY<WorkMinY THEN
                NextY:=WorkMinY;
            ENDIF

            ! Step to next Y row
            pPanEnd.trans.y:=NextY;
            MoveL pPanEnd,vPanTravel,z5,tHeli\WObj:=Bed1Wyong;
            CurrentY:=NextY;

            ! Flip sweep direction
            SweepDir:=-SweepDir;
            IF SweepDir=1 THEN
                StartX:=WorkMinX;
                EndX:=WorkMaxX;
            ELSE
                StartX:=WorkMaxX;
                EndX:=WorkMinX;
            ENDIF

            ! Set up end position for next sweep
            pPanEnd.trans.x:=-EndX;
            pPanEnd.extax.eax_a:=Bed1Wyong.uframe.trans.x-EndX;
        ENDWHILE

        ! ========== PASS 2: Y-direction sweeps (stepping in X) ==========

        ! Reset for Y-direction passes - start from current position
        CurrentX:=Abs(pPanEnd.trans.x);

        ! Determine step direction based on where Pass 1 ended
        ! At high X, step toward low X; at low X, step toward high X
        IF CurrentX>((WorkMinX+WorkMaxX)/2) THEN
            StepDir:=-1;
        ELSE
            StepDir:=1;
        ENDIF

        SweepDir:=1;
        StartY:=WorkMaxY;
        EndY:=WorkMinY;

        ! Set up for Y sweep and move to start position
        pPanEnd.trans.y:=EndY;
        MoveL pPanEnd,vPanTravel,z5,tHeli\WObj:=Bed1Wyong;

        WHILE TRUE DO
            ! Calculate next column
            NextX:=CurrentX+(StepDir*StepSize);

            ! Check if pass complete
            IF (StepDir=1 AND NextX>WorkMaxX) OR (StepDir=-1 AND NextX<WorkMinX) THEN
                EXIT;
            ENDIF

            ! Clamp to bounds
            IF NextX>WorkMaxX THEN
                NextX:=WorkMaxX;
            ELSEIF NextX<WorkMinX THEN
                NextX:=WorkMinX;
            ENDIF

            ! Step to next X column
            pPanEnd.trans.x:=-NextX;
            pPanEnd.extax.eax_a:=Bed1Wyong.uframe.trans.x-NextX;
            MoveL pPanEnd,vPanTravel,z5,tHeli\WObj:=Bed1Wyong;
            CurrentX:=NextX;

            ! Flip sweep direction
            SweepDir:=-SweepDir;
            IF SweepDir=1 THEN
                StartY:=WorkMinY;
                EndY:=WorkMaxY;
            ELSE
                StartY:=WorkMaxY;
                EndY:=WorkMinY;
            ENDIF

            ! Set up end position for next sweep
            pPanEnd.trans.y:=EndY;

            ! === SWEEP Y (full length) ===
            MoveL pPanEnd,vPanTravel,z5,tHeli\WObj:=Bed1Wyong;
        ENDWHILE

        ! === LIFT OFF BED ===
        pPanPos.trans.z:=SafeZ;
        MoveL pPanPos,v100,z5,tHeli\WObj:=Bed1Wyong;

        ! === STOP BLADE ROTATION ===
        HeliBladeSpeed 0,"FWD";
        WaitTime\InPos,3;

        ConfL\On;
        ConfJ\On;

        ! === PACKAWAY ===
        Heli_Dropoff;
        Home;

        TPWrite "PyPan Complete";
    ENDPROC



    ! ========== PY2 GENERATED PROCEDURES ==========
    ! Generated: 05-feb_13:54
    ! Do not edit manually - regenerate via web interface


    PROC Py2Main()
        ! Py2Main - Python-generated tools menu
        ! Generated: 05-feb_13:54

        VAR num iChoice;

        TPErase;
        TPWrite "=== Py2 Tools (05-feb_13:54) ===";
        TPWrite "Panel X: " \Num:=5000;
        TPWrite "Panel Y: " \Num:=1600;
        TPReadNum iChoice,"1:Heli,2:Polish,3:Vacuum";

        TEST iChoice
        CASE 1:
            Py2Heli;
        CASE 2:
            Py2Polish;
        CASE 3:
            Py2Vacuum;
        DEFAULT:
            TPWrite "Invalid choice";
        ENDTEST
    ENDPROC



    PROC Py2Heli()
        ! Py2Heli - Cross-hatch pattern (Andrew's pattern base)
        ! Generated by Onyx Toolpath Generator v2
        ! Panel: (2350,200) to (7350,1800)
        ! Z = FormHeight(150) + z_offset(150) = 300mm
        ! Step: 350mm
        ! Pattern: X passes first, then Y passes

        VAR robtarget pStart;
        VAR robtarget pEnd;
        VAR robtarget pCurrent;
        VAR jointtarget CurrentJoints;
        VAR robtarget CurrentPos;
        VAR num WorkZ:=0;
        VAR num SafeZ:=0;
        VAR num CurrentY:=0;
        VAR num CurrentX:=0;
        VAR num MinY:=0;
        VAR num MaxY:=0;
        VAR num MinX:=0;
        VAR num MaxX:=0;
        VAR num StepSize:=350;
        VAR num SweepDir:=1;
        VAR num StepDir:=1;
        VAR num PassCount:=0;
        VAR num NextX:=0;
        VAR num StartY:=0;
        VAR num EndY:=0;
        VAR bool bDone:=FALSE;
        VAR speeddata vTravel:=[500,15,2000,15];
        VAR num TrackMin:=-300;
        VAR num TrackMax:=10050;
        VAR num CalcTrack:=0;

        ! Initialize runtime values
        WorkZ:=FormHeight+150;
        SafeZ:=WorkZ+200;
        MinY:=200+600/2;
        MaxY:=1800-600/2;
        MinX:=2350+600/2;
        MaxX:=7350-600/2;

        TPWrite "========================================";
        TPWrite "Py2Heli: Cross-hatch Starting";
        TPWrite "========================================";
        TPWrite "Panel X: " \Num:=2350;
        TPWrite " to X: " \Num:=7350;
        TPWrite "Panel Y: " \Num:=200;
        TPWrite " to Y: " \Num:=1800;
        TPWrite "WorkZ=" \Num:=WorkZ;
        TPWrite "SafeZ=" \Num:=SafeZ;
        TPWrite "MinX=" \Num:=MinX;
        TPWrite "MaxX=" \Num:=MaxX;
        TPWrite "MinY=" \Num:=MinY;
        TPWrite "MaxY=" \Num:=MaxY;
        TPWrite "StepSize=" \Num:=StepSize;

        ! Get helicopter if needed
        IF ToolNum<>2 THEN
            TPWrite "Py2Heli: Getting helicopter...";
            Home;
            Heli_Pickup;
        ENDIF

        ! ============================================
        ! PHASE 1: X PASSES (sweep X, step in Y)
        ! Start at far Y, work back toward track
        ! ============================================
        TPWrite "========================================";
        TPWrite "=== PHASE 1: X Passes ===";
        TPWrite "========================================";
        CurrentY:=MaxY;
        SweepDir:=1;
        PassCount:=0;
        TPWrite "P1: Starting at CurrentY=" \Num:=CurrentY;
        TPWrite "P1: Will step toward MinY=" \Num:=MinY;

        ! Initialize start position (X negated per Andrew's pattern)
        pStart.trans:=[-1*(MinX-100),CurrentY,WorkZ];
        pStart.rot:=OrientZYX(0,0,180);
        pStart.robconf:=[0,0,0,0];

        IF CurrentY<1800 THEN
            CalcTrack:=Bed1Wyong.uframe.trans.x+pStart.trans.x+1000+600/2;
        ELSE
            CalcTrack:=Bed1Wyong.uframe.trans.x+pStart.trans.x+600/2;
        ENDIF
        IF CalcTrack<TrackMin THEN CalcTrack:=TrackMin; ENDIF
        IF CalcTrack>TrackMax THEN CalcTrack:=TrackMax; ENDIF
        pStart.extax:=[CalcTrack,9E+09,9E+09,9E+09,9E+09,9E+09];

        pEnd:=pStart;
        pEnd.trans.x:=-1*(MaxX+100);
        IF CurrentY<1800 THEN
            CalcTrack:=Bed1Wyong.uframe.trans.x+pEnd.trans.x+1000-600/2;
        ELSE
            CalcTrack:=Bed1Wyong.uframe.trans.x+pEnd.trans.x-600/2;
        ENDIF
        IF CalcTrack<TrackMin THEN CalcTrack:=TrackMin; ENDIF
        IF CalcTrack>TrackMax THEN CalcTrack:=TrackMax; ENDIF
        pEnd.extax.eax_a:=CalcTrack;

        ! Move to start position (safe height)
        pStart.trans.z:=SafeZ;
        MoveJ pStart,v500,z5,tHeli\WObj:=Bed1Wyong;

        ! Home stepper and set blade angle
        TPWrite "Py2Heli: Homing stepper...";
        Heli_Stepper_Home;
        HeliBlade_Angle 0;
        WaitTime 1;

        ! Disable configuration tracking for cross-hatch movements
        ConfL\Off;
        ConfJ\Off;

        ! Start blade rotation
        TPWrite "Py2Heli: Starting blade...";
        HeliBladeSpeed 70,"FWD";
        WaitTime 2;

        ! Lower to work height
        pStart.trans.z:=WorkZ;
        MoveJ Offs(pStart,0,0,50),v100,z5,tHeli\WObj:=Bed1Wyong;
        MoveL pStart,v50,fine,tHeli\WObj:=Bed1Wyong;

        TPWrite "P1: Entering X-pass loop...";
        bDone:=FALSE;

        ! X-pass loop (using flag instead of EXIT)
        WHILE CurrentY>=MinY AND bDone=FALSE DO
            Incr PassCount;
            TPWrite "----------------------------------------";
            TPWrite "P1: X Pass " \Num:=PassCount;
            TPWrite "P1: CurrentY=" \Num:=CurrentY;
            TPWrite "P1: SweepDir=" \Num:=SweepDir;

            pStart.trans.y:=CurrentY;
            pEnd.trans.y:=CurrentY;

            IF CurrentY<1800 THEN
                CalcTrack:=Bed1Wyong.uframe.trans.x+pStart.trans.x+1000+600/2;
            ELSE
                CalcTrack:=Bed1Wyong.uframe.trans.x+pStart.trans.x+600/2;
            ENDIF
            IF CalcTrack<TrackMin THEN CalcTrack:=TrackMin; ENDIF
            IF CalcTrack>TrackMax THEN CalcTrack:=TrackMax; ENDIF
            pStart.extax.eax_a:=CalcTrack;

            IF CurrentY<1800 THEN
                CalcTrack:=Bed1Wyong.uframe.trans.x+pEnd.trans.x+1000-600/2;
            ELSE
                CalcTrack:=Bed1Wyong.uframe.trans.x+pEnd.trans.x-600/2;
            ENDIF
            IF CalcTrack<TrackMin THEN CalcTrack:=TrackMin; ENDIF
            IF CalcTrack>TrackMax THEN CalcTrack:=TrackMax; ENDIF
            pEnd.extax.eax_a:=CalcTrack;

            IF SweepDir=1 THEN
                TPWrite "P1: Sweep to pEnd (far X)";
                MoveL pEnd,vTravel,fine,tHeli\WObj:=Bed1Wyong;
            ELSE
                TPWrite "P1: Sweep to pStart (near X)";
                MoveL pStart,vTravel,fine,tHeli\WObj:=Bed1Wyong;
            ENDIF
            TPWrite "P1: Sweep complete";

            IF (CurrentY-StepSize)<MinY THEN
                TPWrite "P1: Last pass - (CurrentY-StepSize) < MinY";
                TPWrite "P1: Setting bDone=TRUE to exit loop";
                bDone:=TRUE;
            ELSE
                ! Only step to next row if not done
                CurrentY:=CurrentY-StepSize;
                TPWrite "P1: Step to next Y row=" \Num:=CurrentY;

                IF SweepDir=1 THEN
                    pEnd.trans.y:=CurrentY;
                    IF CurrentY<1800 THEN
                        CalcTrack:=Bed1Wyong.uframe.trans.x+pEnd.trans.x+1000-600/2;
                    ELSE
                        CalcTrack:=Bed1Wyong.uframe.trans.x+pEnd.trans.x-600/2;
                    ENDIF
                    IF CalcTrack<TrackMin THEN CalcTrack:=TrackMin; ENDIF
                    IF CalcTrack>TrackMax THEN CalcTrack:=TrackMax; ENDIF
                    pEnd.extax.eax_a:=CalcTrack;
                    MoveL pEnd,vTravel,fine,tHeli\WObj:=Bed1Wyong;
                ELSE
                    pStart.trans.y:=CurrentY;
                    IF CurrentY<1800 THEN
                        CalcTrack:=Bed1Wyong.uframe.trans.x+pStart.trans.x+1000+600/2;
                    ELSE
                        CalcTrack:=Bed1Wyong.uframe.trans.x+pStart.trans.x+600/2;
                    ENDIF
                    IF CalcTrack<TrackMin THEN CalcTrack:=TrackMin; ENDIF
                    IF CalcTrack>TrackMax THEN CalcTrack:=TrackMax; ENDIF
                    pStart.extax.eax_a:=CalcTrack;
                    MoveL pStart,vTravel,fine,tHeli\WObj:=Bed1Wyong;
                ENDIF

                SweepDir:=-1*SweepDir;
            ENDIF
        ENDWHILE

        TPWrite "P1: X passes complete, total=" \Num:=PassCount;
        TPWrite "P1: Final position Y=" \Num:=CurrentY;
        TPWrite "P1: pEnd.trans.x=" \Num:=pEnd.trans.x;

        ! ============================================
        ! PHASE 2: Y PASSES (sweep Y, step in X)
        ! Continue from where Pass 1 ended (like baseline PyHeli)
        ! ============================================
        TPWrite "========================================";
        TPWrite "=== PHASE 2: Y Passes ===";
        TPWrite "========================================";

        ! Continue from where X passes ended - NO diagonal repositioning
        ! Determine actual X position based on final sweep direction
        IF SweepDir=1 THEN
            ! Last sweep was forward, so we ended at MaxX
            CurrentX:=MaxX;
        ELSE
            ! Last sweep was reverse, so we ended at MinX
            CurrentX:=MinX;
        ENDIF
        TPWrite "P2: Starting from CurrentX=" \Num:=CurrentX;
        TPWrite "P2: Starting from CurrentY=" \Num:=CurrentY;

        ! Step direction: continue stepping in X from where we are
        IF CurrentX>=MaxX THEN
            StepDir:=-1;
            TPWrite "P2: StepDir=-1 (toward MinX)";
        ELSE
            StepDir:=1;
            TPWrite "P2: StepDir=+1 (toward MaxX)";
        ENDIF

        ! First Y sweep: go to opposite Y bound from current position
        ! This is just a straight Y move, no X change
        IF CurrentY>((MinY+MaxY)/2) THEN
            EndY:=MinY;
            TPWrite "P2: First sweep toward MinY";
        ELSE
            EndY:=MaxY;
            TPWrite "P2: First sweep toward MaxY";
        ENDIF

        PassCount:=0;

        ! First Y sweep from current position (straight Y move, no diagonal)
        TPWrite "P2: First Y sweep to EndY=" \Num:=EndY;
        pEnd.trans.x:=-1*CurrentX;
        pEnd.trans.y:=EndY;
        TPWrite "P2: Moving...";
        MoveL pEnd,vTravel,fine,tHeli\WObj:=Bed1Wyong;
        CurrentY:=EndY;
        TPWrite "P2: First Y sweep complete";

        TPWrite "P2: Entering Y-pass loop...";
        bDone:=FALSE;

        ! Y-pass loop - step in X, sweep in Y (using flag instead of EXIT)
        WHILE bDone=FALSE DO
            Incr PassCount;
            TPWrite "----------------------------------------";
            TPWrite "P2: Y Pass " \Num:=PassCount;

            ! Calculate next column
            NextX:=CurrentX+(StepDir*StepSize);
            TPWrite "P2: CurrentX=" \Num:=CurrentX;
            TPWrite "P2: NextX=" \Num:=NextX;

            ! Check if complete
            IF (StepDir=1 AND NextX>MaxX) OR (StepDir=-1 AND NextX<MinX) THEN
                TPWrite "P2: NextX out of bounds - setting bDone=TRUE";
                bDone:=TRUE;
            ELSE
                ! Clamp to bounds
                IF NextX>MaxX THEN
                    NextX:=MaxX;
                    TPWrite "P2: Clamped to MaxX";
                ELSEIF NextX<MinX THEN
                    NextX:=MinX;
                    TPWrite "P2: Clamped to MinX";
                ENDIF

                ! Step to next X column
                TPWrite "P2: Step to X=" \Num:=NextX;
                pEnd.trans.x:=-1*NextX;
                CalcTrack:=Bed1Wyong.uframe.trans.x-NextX;
                IF CalcTrack<TrackMin THEN CalcTrack:=TrackMin; ENDIF
                IF CalcTrack>TrackMax THEN CalcTrack:=TrackMax; ENDIF
                pEnd.extax.eax_a:=CalcTrack;
                TPWrite "P2: Moving to next X column...";
                MoveL pEnd,vTravel,fine,tHeli\WObj:=Bed1Wyong;
                TPWrite "P2: Step complete";
                CurrentX:=NextX;

                ! Flip sweep direction
                SweepDir:=-1*SweepDir;
                IF SweepDir=1 THEN
                    EndY:=MinY;
                    TPWrite "P2: Next sweep toward MinY=" \Num:=EndY;
                ELSE
                    EndY:=MaxY;
                    TPWrite "P2: Next sweep toward MaxY=" \Num:=EndY;
                ENDIF

                ! Sweep Y
                TPWrite "P2: Sweep to Y=" \Num:=EndY;
                pEnd.trans.y:=EndY;
                TPWrite "P2: Moving...";
                MoveL pEnd,vTravel,fine,tHeli\WObj:=Bed1Wyong;
                TPWrite "P2: Sweep complete";
            ENDIF
        ENDWHILE

        TPWrite "========================================";
        TPWrite "P2: Y passes complete, total=" \Num:=PassCount;
        TPWrite "Cross-hatch complete!";
        TPWrite "========================================";

        ! ============================================
        ! FINISH: Stop blade, lift tool, return
        ! ============================================
        TPWrite "========================================";
        TPWrite "=== FINISH ===";
        TPWrite "========================================";

        TPWrite "FINISH: Stopping blade...";
        HeliBladeSpeed 0,"FWD";
        WaitTime 1;
        TPWrite "FINISH: Blade stopped";

        ! Lift off the bed
        TPWrite "FINISH: Lifting off bed...";
        CurrentJoints:=CJointT();
        CurrentPos:=CalcRobT(CurrentJoints,tHeli\WObj:=Bed1Wyong);
        MoveJ Offs(CurrentPos,0,0,200),v100,fine,tHeli\WObj:=Bed1Wyong;
        TPWrite "FINISH: Lifted 200mm";

        ! Re-enable configuration tracking
        TPWrite "FINISH: Re-enabling ConfL/ConfJ...";
        ConfL\On;
        ConfJ\On;
        TPWrite "FINISH: Configuration tracking enabled";

        ! Return tool
        TPWrite "FINISH: Dropping off helicopter...";
        Heli_Dropoff;
        TPWrite "FINISH: Helicopter dropped off";

        TPWrite "FINISH: Homing...";
        Home;

        TPWrite "========================================";
        TPWrite "Py2Heli: COMPLETE";
        TPWrite "========================================";

    ERROR
        HeliBladeSpeed 0,"FWD";
        RAISE;
    ENDPROC



    PROC Py2Polish()
        ! Py2Polish - Polisher with force control
        ! Generated by Onyx Toolpath Generator v2
        ! Workzone: bed
        ! First direction: x
        ! Area: (225,225) to (2500,1650)
        ! Z = 50mm (FormHeight + offset)
        ! Step: 450mm
        ! Force: Start=200N, Motion=200N

        VAR robtarget pStart;
        VAR robtarget pEnd;
        VAR jointtarget CurrentJoints;
        VAR robtarget CurrentPos;
        VAR num WorkZ:=0;
        VAR num SafeZ:=0;
        VAR num CurrentY:=0;
        VAR num MinY:=0;
        VAR num MaxY:=0;
        VAR num MinX:=0;
        VAR num MaxX:=0;
        VAR num StepSize:=450;
        VAR num SweepDir:=1;
        VAR num StepDir:=1;
        VAR num PassCount:=0;
        VAR bool bDone:=FALSE;
        VAR num CurrentX:=0;
        VAR num StartY:=0;
        VAR num EndY:=0;
        VAR num NextX:=0;
        VAR speeddata vApproach:=[20,15,2000,15];
        VAR speeddata vRetract:=[50,15,2000,15];
        VAR speeddata vTravel:=[100,15,2000,15];
        VAR num TrackMin:=-300;
        VAR num TrackMax:=10050;
        VAR num CalcTrack:=0;

        ! Initialize runtime values
        WorkZ:=50;
        SafeZ:=WorkZ+200;
        MinY:=225;
        MaxY:=1650;
        MinX:=225;
        MaxX:=2500;

        TPWrite "========================================";
        TPWrite "Py2Polish: Starting";
        TPWrite "========================================";
        TPWrite "Workzone: bed";
        TPWrite "MinX=" \Num:=MinX;
        TPWrite "MaxX=" \Num:=MaxX;
        TPWrite "MinY=" \Num:=MinY;
        TPWrite "MaxY=" \Num:=MaxY;
        TPWrite "WorkZ=" \Num:=WorkZ;
        TPWrite "StepSize=" \Num:=StepSize;
        TPWrite "Force Control: ENABLED";

        ! Get polisher if needed
        IF ToolNum<>6 THEN
            TPWrite "Py2Polish: Getting polisher...";
            Home;
            Polish_Pickup;
        ELSE
            ! Already have polisher - ensure safe height
            CurrentJoints:=CJointT();
            CurrentPos:=CalcRobT(CurrentJoints,tPolish\WObj:=wobj0);
            IF CurrentPos.trans.z<600 THEN
                MoveL Offs(CurrentPos,0,0,(600-CurrentPos.trans.z)),v500,z5,tPolish;
            ENDIF
        ENDIF

        ! ============================================
        ! PHASE 1: X PASSES (sweep X, step in Y)
        ! First direction: x
        ! ============================================
        CurrentY:=MaxY;
        SweepDir:=1;
        PassCount:=0;

        TPWrite "Cross-hatch, first direction: x";
        TPWrite "Starting P1 (X passes) at Y=" \Num:=CurrentY;

        ! Initialize start position (X negated per Andrew's pattern)
        pStart.trans:=[-1*MinX,CurrentY,SafeZ];
        pStart.rot:=OrientZYX(0,0,180);
        pStart.robconf:=[0,0,0,0];

        ! Clamp track position to limits - arm will extend to reach target
        CalcTrack:=Bed1Wyong.uframe.trans.x+pStart.trans.x;
        IF CalcTrack<TrackMin THEN CalcTrack:=TrackMin; ENDIF
        IF CalcTrack>TrackMax THEN CalcTrack:=TrackMax; ENDIF
        pStart.extax:=[CalcTrack,9E+09,9E+09,9E+09,9E+09,9E+09];

        pEnd:=pStart;
        pEnd.trans.x:=-1*MaxX;
        CalcTrack:=Bed1Wyong.uframe.trans.x+pEnd.trans.x;
        IF CalcTrack<TrackMin THEN CalcTrack:=TrackMin; ENDIF
        IF CalcTrack>TrackMax THEN CalcTrack:=TrackMax; ENDIF
        pEnd.extax.eax_a:=CalcTrack;

        ! Move to start position (safe height)
        MoveJ pStart,v500,z5,tPolish\WObj:=Bed1Wyong;

        ! Disable configuration tracking
        ConfL\Off;
        ConfJ\Off;

        ! Turn on polisher (only if force control enabled)
        Pol_on;

        ! Lower to work height and START force control ONCE before cross-hatch
        pStart.trans.z:=WorkZ;
        pEnd.trans.z:=WorkZ;
        MoveJ Offs(pStart,0,0,50),v100,z5,tPolish\WObj:=Bed1Wyong;

        ! Start force control - stays active for entire cross-hatch
        WaitTime\inpos,0.1;
        FCCalib PolishLoad;
        FCPress1LStart pStart,vApproach,\Fz:=200,15,\ForceChange:=150\PosSupvDist:=100,z5,tPolish\WObj:=Bed1Wyong;

        TPWrite "On work surface, starting cross-hatch...";

        bDone:=FALSE;

        ! X-pass loop - STAY ON SURFACE throughout
        WHILE CurrentY>=MinY AND bDone=FALSE DO
            Incr PassCount;
            TPWrite "----------------------------------------";
            TPWrite "Pass " \Num:=PassCount;
            TPWrite "CurrentY=" \Num:=CurrentY;
            TPWrite "SweepDir=" \Num:=SweepDir;

            ! Update Y position (Z stays at WorkZ)
            pStart.trans.y:=CurrentY;
            pEnd.trans.y:=CurrentY;

            IF SweepDir=1 THEN
                ! Forward pass (MinX to MaxX) - stay on surface with force control
                TPWrite "Forward pass to MaxX";
                FCPressL pEnd,vTravel,200,fine,tPolish\WObj:=Bed1Wyong;
            ELSE
                ! Reverse pass (MaxX to MinX) - stay on surface with force control
                TPWrite "Reverse pass to MinX";
                FCPressL pStart,vTravel,200,fine,tPolish\WObj:=Bed1Wyong;
            ENDIF

            TPWrite "Pass complete";

            ! Check if we should continue
            IF (CurrentY-StepSize)<MinY THEN
                TPWrite "Last pass reached - done";
                bDone:=TRUE;
            ELSE
                ! Step to next row - STAY ON SURFACE
                CurrentY:=CurrentY-StepSize;
                TPWrite "Step to Y=" \Num:=CurrentY;

                ! Update Y and step while staying on surface (clamp track to limits)
                IF SweepDir=1 THEN
                    pEnd.trans.y:=CurrentY;
                    CalcTrack:=Bed1Wyong.uframe.trans.x+pEnd.trans.x;
                    IF CalcTrack<TrackMin THEN CalcTrack:=TrackMin; ENDIF
                    IF CalcTrack>TrackMax THEN CalcTrack:=TrackMax; ENDIF
                    pEnd.extax.eax_a:=CalcTrack;
                    FCPressL pEnd,vTravel,200,fine,tPolish\WObj:=Bed1Wyong;
                ELSE
                    pStart.trans.y:=CurrentY;
                    CalcTrack:=Bed1Wyong.uframe.trans.x+pStart.trans.x;
                    IF CalcTrack<TrackMin THEN CalcTrack:=TrackMin; ENDIF
                    IF CalcTrack>TrackMax THEN CalcTrack:=TrackMax; ENDIF
                    pStart.extax.eax_a:=CalcTrack;
                    FCPressL pStart,vTravel,200,fine,tPolish\WObj:=Bed1Wyong;
                ENDIF

                ! Flip direction
                SweepDir:=-1*SweepDir;
            ENDIF
        ENDWHILE

        TPWrite "P1: X passes complete, total=" \Num:=PassCount;

        ! ============================================
        ! PHASE 2: Y PASSES (sweep Y, step in X)
        ! Cross-hatch pattern - continue from Phase 1
        ! ============================================
        TPWrite "========================================";
        TPWrite "=== PHASE 2: Y Passes ===";
        TPWrite "========================================";

        ! Continue from where X passes ended - NO diagonal repositioning
        ! Determine actual X position based on final sweep direction
        IF SweepDir=1 THEN
            ! Last sweep was forward, so we ended at MaxX
            CurrentX:=MaxX;
        ELSE
            ! Last sweep was reverse, so we ended at MinX
            CurrentX:=MinX;
        ENDIF
        TPWrite "P2: Starting from CurrentX=" \Num:=CurrentX;
        TPWrite "P2: Starting from CurrentY=" \Num:=CurrentY;

        ! Step direction: continue stepping in X from where we are
        IF CurrentX>=MaxX THEN
            StepDir:=-1;
            TPWrite "P2: StepDir=-1 (toward MinX)";
        ELSE
            StepDir:=1;
            TPWrite "P2: StepDir=+1 (toward MaxX)";
        ENDIF

        ! First Y sweep: go to opposite Y bound from current position
        IF CurrentY>((MinY+MaxY)/2) THEN
            EndY:=MinY;
            TPWrite "P2: First sweep toward MinY";
        ELSE
            EndY:=MaxY;
            TPWrite "P2: First sweep toward MaxY";
        ENDIF

        PassCount:=0;

        ! First Y sweep from current position (straight Y move, no diagonal)
        TPWrite "P2: First Y sweep to EndY=" \Num:=EndY;
        pEnd.trans.x:=-1*CurrentX;
        pEnd.trans.y:=EndY;
        TPWrite "P2: Moving...";
        FCPressL pEnd,vTravel,200,fine,tPolish\WObj:=Bed1Wyong;
        CurrentY:=EndY;
        TPWrite "P2: First Y sweep complete";

        TPWrite "P2: Entering Y-pass loop...";
        bDone:=FALSE;

        ! Y-pass loop - step in X, sweep in Y
        WHILE bDone=FALSE DO
            Incr PassCount;
            TPWrite "----------------------------------------";
            TPWrite "P2: Y Pass " \Num:=PassCount;

            ! Calculate next column
            NextX:=CurrentX+(StepDir*StepSize);
            TPWrite "P2: CurrentX=" \Num:=CurrentX;
            TPWrite "P2: NextX=" \Num:=NextX;

            ! Check if complete
            IF (StepDir=1 AND NextX>MaxX) OR (StepDir=-1 AND NextX<MinX) THEN
                TPWrite "P2: NextX out of bounds - done";
                bDone:=TRUE;
            ELSE
                ! Clamp to bounds
                IF NextX>MaxX THEN
                    NextX:=MaxX;
                    TPWrite "P2: Clamped to MaxX";
                ELSEIF NextX<MinX THEN
                    NextX:=MinX;
                    TPWrite "P2: Clamped to MinX";
                ENDIF

                ! Step to next X column (stay on surface)
                TPWrite "P2: Step to X=" \Num:=NextX;
                pEnd.trans.x:=-1*NextX;
                CalcTrack:=Bed1Wyong.uframe.trans.x+pEnd.trans.x;
                IF CalcTrack<TrackMin THEN CalcTrack:=TrackMin; ENDIF
                IF CalcTrack>TrackMax THEN CalcTrack:=TrackMax; ENDIF
                pEnd.extax.eax_a:=CalcTrack;
                TPWrite "P2: Moving to next X column...";
                FCPressL pEnd,vTravel,200,fine,tPolish\WObj:=Bed1Wyong;
                TPWrite "P2: Step complete";
                CurrentX:=NextX;

                ! Flip sweep direction
                SweepDir:=-1*SweepDir;
                IF SweepDir=1 THEN
                    EndY:=MinY;
                    TPWrite "P2: Next sweep toward MinY=" \Num:=EndY;
                ELSE
                    EndY:=MaxY;
                    TPWrite "P2: Next sweep toward MaxY=" \Num:=EndY;
                ENDIF

                ! Sweep Y
                TPWrite "P2: Sweep to Y=" \Num:=EndY;
                pEnd.trans.y:=EndY;
                TPWrite "P2: Moving...";
                FCPressL pEnd,vTravel,200,fine,tPolish\WObj:=Bed1Wyong;
                TPWrite "P2: Sweep complete";
            ENDIF
        ENDWHILE

        TPWrite "========================================";
        TPWrite "P2: Y passes complete, total=" \Num:=PassCount;
        TPWrite "Cross-hatch complete!";
        TPWrite "========================================";

        ! END force control ONCE after all passes complete
        CurrentJoints:=CJointT();
        CurrentPos:=CalcRobT(CurrentJoints,tPolish\WObj:=Bed1Wyong);
        FCPressEnd Offs(CurrentPos,0,0,75),vRetract,\DeactOnly,tPolish\WObj:=Bed1Wyong;

        TPWrite "========================================";
        TPWrite "Py2Polish: Complete";
        TPWrite "Total passes=" \Num:=PassCount;
        TPWrite "========================================";

        ! Ensure polisher is off (only if it was turned on)
        Pol_off;

        ! Re-enable configuration tracking
        ConfL\On;
        ConfJ\On;

        ! Return to safe position (already lifted if force control was used)
        ! Already lifted by FCPressEnd
        ! Moving to safe height


        ! Return tool and go home
        TPWrite "Py2Polish: Dropping off polisher...";
        Polish_Dropoff;
        TPWrite "Py2Polish: Polisher dropped off";

        TPWrite "Py2Polish: Homing...";
        Home;

        TPWrite "========================================";
        TPWrite "Py2Polish: COMPLETE";
        TPWrite "========================================";

    ERROR
        Pol_off;
        TPWrite "Py2Polish ERROR: " \Num:=ERRNO;
        RAISE;
    ENDPROC



    PROC Py2Vacuum()
        ! Py2Vacuum - Cross-hatch pattern for vacuum
        ! Generated by Onyx Toolpath Generator v2
        ! Workzone: bed
        ! Area: (0,0) to (2500,1650)
        ! Z = -20mm
        ! Step: 300mm
        ! Pattern: X passes first, then Y passes

        VAR robtarget pStart;
        VAR robtarget pEnd;
        VAR jointtarget CurrentJoints;
        VAR robtarget CurrentPos;
        VAR num WorkZ:=0;
        VAR num SafeZ:=0;
        VAR num CurrentY:=0;
        VAR num CurrentX:=0;
        VAR num MinY:=0;
        VAR num MaxY:=0;
        VAR num MinX:=0;
        VAR num MaxX:=0;
        VAR num StepSize:=300;
        VAR num SweepDir:=1;
        VAR num StepDir:=1;
        VAR num PassCount:=0;
        VAR num NextX:=0;
        VAR num StartY:=0;
        VAR num EndY:=0;
        VAR bool bDone:=FALSE;
        VAR speeddata vTravel:=[200,15,2000,15];
        VAR num TrackMin:=-300;
        VAR num TrackMax:=10050;
        VAR num CalcTrack:=0;

        ! Initialize runtime values
        WorkZ:=-20;
        SafeZ:=WorkZ+200;
        MinY:=0+400/2;
        MaxY:=1650-400/2;
        MinX:=0+400/2;
        MaxX:=2500-400/2;

        TPWrite "========================================";
        TPWrite "Py2Vacuum: Cross-hatch Starting";
        TPWrite "========================================";
        TPWrite "Workzone: bed";
        TPWrite "MinX=" \Num:=MinX;
        TPWrite "MaxX=" \Num:=MaxX;
        TPWrite "MinY=" \Num:=MinY;
        TPWrite "MaxY=" \Num:=MaxY;
        TPWrite "WorkZ=" \Num:=WorkZ;
        TPWrite "StepSize=" \Num:=StepSize;

        ! Get vacuum if needed
        IF ToolNum<>5 THEN
            TPWrite "Py2Vacuum: Getting vacuum...";
            Home;
            Vac_Pickup;
        ELSE
            ! Already have vacuum - ensure safe height
            CurrentJoints:=CJointT();
            CurrentPos:=CalcRobT(CurrentJoints,tVac\WObj:=Bed1Wyong);
            IF CurrentPos.trans.z<600 THEN
                MoveL Offs(CurrentPos,0,0,(600-CurrentPos.trans.z)),v500,z5,tVac\WObj:=Bed1Wyong;
            ENDIF
        ENDIF

        ! ============================================
        ! PHASE 1: X PASSES (sweep X, step in Y)
        ! Start at far Y (MaxY), work back toward track
        ! ============================================
        TPWrite "P1: Starting X passes...";
        CurrentY:=MaxY;
        SweepDir:=1;
        PassCount:=0;
        TPWrite "P1: Starting at CurrentY=" \Num:=CurrentY;

        ! Initialize start position (X negated per Bed1Wyong)
        pStart.trans:=[-1*(MinX-100),CurrentY,WorkZ];
        pStart.rot:=OrientZYX(0,0,180);
        pStart.robconf:=[0,0,0,0];

        ! Clamp track position
        CalcTrack:=Bed1Wyong.uframe.trans.x+pStart.trans.x+400/2;
        IF CalcTrack<TrackMin THEN CalcTrack:=TrackMin; ENDIF
        IF CalcTrack>TrackMax THEN CalcTrack:=TrackMax; ENDIF
        pStart.extax:=[CalcTrack,9E+09,9E+09,9E+09,9E+09,9E+09];

        pEnd:=pStart;
        pEnd.trans.x:=-1*(MaxX+100);
        CalcTrack:=Bed1Wyong.uframe.trans.x+pEnd.trans.x-400/2;
        IF CalcTrack<TrackMin THEN CalcTrack:=TrackMin; ENDIF
        IF CalcTrack>TrackMax THEN CalcTrack:=TrackMax; ENDIF
        pEnd.extax.eax_a:=CalcTrack;

        ! Move to start position (safe height)
        pStart.trans.z:=SafeZ;
        MoveJ pStart,v500,z5,tVac\WObj:=Bed1Wyong;

        ! Disable configuration tracking
        ConfL\Off;
        ConfJ\Off;

        ! Turn on vacuum
        TPWrite "Py2Vacuum: Starting vacuum...";
        Vac_on;
        WaitTime 1;

        ! Lower to work height
        pStart.trans.z:=WorkZ;
        pEnd.trans.z:=WorkZ;
        MoveJ Offs(pStart,0,0,50),v100,z5,tVac\WObj:=Bed1Wyong;
        MoveL pStart,v50,fine,tVac\WObj:=Bed1Wyong;

        TPWrite "P1: Entering X-pass loop...";
        bDone:=FALSE;

        ! X-pass loop
        WHILE CurrentY>=MinY AND bDone=FALSE DO
            Incr PassCount;
            TPWrite "----------------------------------------";
            TPWrite "P1: X Pass " \Num:=PassCount;
            TPWrite "P1: CurrentY=" \Num:=CurrentY;

            pStart.trans.y:=CurrentY;
            pEnd.trans.y:=CurrentY;

            ! Update extax with clamping
            CalcTrack:=Bed1Wyong.uframe.trans.x+pStart.trans.x+400/2;
            IF CalcTrack<TrackMin THEN CalcTrack:=TrackMin; ENDIF
            IF CalcTrack>TrackMax THEN CalcTrack:=TrackMax; ENDIF
            pStart.extax.eax_a:=CalcTrack;

            CalcTrack:=Bed1Wyong.uframe.trans.x+pEnd.trans.x-400/2;
            IF CalcTrack<TrackMin THEN CalcTrack:=TrackMin; ENDIF
            IF CalcTrack>TrackMax THEN CalcTrack:=TrackMax; ENDIF
            pEnd.extax.eax_a:=CalcTrack;

            IF SweepDir=1 THEN
                TPWrite "P1: Sweep to pEnd (far X)";
                MoveL pEnd,vTravel,fine,tVac\WObj:=Bed1Wyong;
            ELSE
                TPWrite "P1: Sweep to pStart (near X)";
                MoveL pStart,vTravel,fine,tVac\WObj:=Bed1Wyong;
            ENDIF

            IF (CurrentY-StepSize)<MinY THEN
                TPWrite "P1: Last pass - setting bDone=TRUE";
                bDone:=TRUE;
            ELSE
                ! Step to next row
                CurrentY:=CurrentY-StepSize;
                TPWrite "P1: Step to next Y row=" \Num:=CurrentY;

                IF SweepDir=1 THEN
                    pEnd.trans.y:=CurrentY;
                    CalcTrack:=Bed1Wyong.uframe.trans.x+pEnd.trans.x-400/2;
                    IF CalcTrack<TrackMin THEN CalcTrack:=TrackMin; ENDIF
                    IF CalcTrack>TrackMax THEN CalcTrack:=TrackMax; ENDIF
                    pEnd.extax.eax_a:=CalcTrack;
                    MoveL pEnd,vTravel,fine,tVac\WObj:=Bed1Wyong;
                ELSE
                    pStart.trans.y:=CurrentY;
                    CalcTrack:=Bed1Wyong.uframe.trans.x+pStart.trans.x+400/2;
                    IF CalcTrack<TrackMin THEN CalcTrack:=TrackMin; ENDIF
                    IF CalcTrack>TrackMax THEN CalcTrack:=TrackMax; ENDIF
                    pStart.extax.eax_a:=CalcTrack;
                    MoveL pStart,vTravel,fine,tVac\WObj:=Bed1Wyong;
                ENDIF

                SweepDir:=-1*SweepDir;
            ENDIF
        ENDWHILE

        TPWrite "P1: X passes complete, total=" \Num:=PassCount;

        ! ============================================
        ! PHASE 2: Y PASSES (sweep Y, step in X)
        ! Start at current X position, sweep in Y
        ! ============================================
        TPWrite "P2: Starting Y passes...";

        ! Reset for Y passes - start from MinX
        CurrentX:=MinX;
        StepDir:=1;
        PassCount:=0;
        bDone:=FALSE;

        ! Determine sweep direction based on where we ended Phase 1
        IF SweepDir=1 THEN
            StartY:=MinY;
            EndY:=MaxY;
        ELSE
            StartY:=MaxY;
            EndY:=MinY;
        ENDIF

        ! Initialize position for Y sweeps
        pStart.trans:=[-1*CurrentX,StartY,WorkZ];
        pEnd.trans:=[-1*CurrentX,EndY,WorkZ];

        CalcTrack:=Bed1Wyong.uframe.trans.x-CurrentX;
        IF CalcTrack<TrackMin THEN CalcTrack:=TrackMin; ENDIF
        IF CalcTrack>TrackMax THEN CalcTrack:=TrackMax; ENDIF
        pStart.extax.eax_a:=CalcTrack;
        pEnd.extax.eax_a:=CalcTrack;

        TPWrite "P2: Starting at X=" \Num:=CurrentX;
        TPWrite "P2: StartY=" \Num:=StartY;
        TPWrite "P2: EndY=" \Num:=EndY;

        ! Y-pass loop
        WHILE bDone=FALSE DO
            Incr PassCount;
            TPWrite "----------------------------------------";
            TPWrite "P2: Y Pass " \Num:=PassCount;
            TPWrite "P2: CurrentX=" \Num:=CurrentX;

            ! Sweep in Y direction
            IF SweepDir=1 THEN
                TPWrite "P2: Sweep toward MaxY";
                MoveL pEnd,vTravel,fine,tVac\WObj:=Bed1Wyong;
            ELSE
                TPWrite "P2: Sweep toward MinY";
                MoveL pStart,vTravel,fine,tVac\WObj:=Bed1Wyong;
            ENDIF

            ! Calculate next X position
            NextX:=CurrentX+(StepDir*StepSize);

            ! Check if complete
            IF (StepDir=1 AND NextX>MaxX) OR (StepDir=-1 AND NextX<MinX) THEN
                TPWrite "P2: NextX out of bounds - setting bDone=TRUE";
                bDone:=TRUE;
            ELSE
                ! Clamp to bounds
                IF NextX>MaxX THEN
                    NextX:=MaxX;
                ELSEIF NextX<MinX THEN
                    NextX:=MinX;
                ENDIF

                ! Step to next X column
                TPWrite "P2: Step to X=" \Num:=NextX;
                pEnd.trans.x:=-1*NextX;
                pStart.trans.x:=-1*NextX;
                CalcTrack:=Bed1Wyong.uframe.trans.x-NextX;
                IF CalcTrack<TrackMin THEN CalcTrack:=TrackMin; ENDIF
                IF CalcTrack>TrackMax THEN CalcTrack:=TrackMax; ENDIF
                pEnd.extax.eax_a:=CalcTrack;
                pStart.extax.eax_a:=CalcTrack;

                IF SweepDir=1 THEN
                    MoveL pEnd,vTravel,fine,tVac\WObj:=Bed1Wyong;
                ELSE
                    MoveL pStart,vTravel,fine,tVac\WObj:=Bed1Wyong;
                ENDIF

                CurrentX:=NextX;
                SweepDir:=-1*SweepDir;
            ENDIF
        ENDWHILE

        TPWrite "P2: Y passes complete, total=" \Num:=PassCount;

        ! ============================================
        ! FINISH: Turn off vacuum, raise, dropoff
        ! ============================================
        TPWrite "========================================";
        TPWrite "Py2Vacuum: Complete";
        TPWrite "========================================";

        ! Turn off vacuum
        Vac_off;

        ! Raise to safe height
        CurrentJoints:=CJointT();
        CurrentPos:=CalcRobT(CurrentJoints,tVac\WObj:=Bed1Wyong);
        MoveL Offs(CurrentPos,0,0,200),v200,z5,tVac\WObj:=Bed1Wyong;

        ! Re-enable config tracking
        ConfL\On;
        ConfJ\On;

        ! Return tool and go home
        TPWrite "Py2Vacuum: Dropping off vacuum...";
        Vac_Dropoff;
        TPWrite "Py2Vacuum: Vacuum dropped off";

        TPWrite "Py2Vacuum: Homing...";
        Home;

        TPWrite "========================================";
        TPWrite "Py2Vacuum: COMPLETE";
        TPWrite "========================================";

    ERROR
        Vac_off;
        TPWrite "Py2Vacuum ERROR: " \Num:=ERRNO;
        RAISE;
    ENDPROC


    ! ========== END PY2 GENERATED PROCEDURES ==========

ENDMODULE
